(* IEC 61131-3 sources: std_i2980_v2.06_cp053/Source/IMM/ieccontrol/EjectorGeneral, 15 files *)

(* ---- FBConvertLintab.pu ---- *)
(*
@h    ! WARNING !
@h    The Kemro K2 system (including software) only meets category B according to EN 954-1,
@h    thus it is not intended for usage in safety-relevant control applications in the field
@h    of personal safety (e.g. emergency stop).
@h    To implement potentially necessary safety-relevant control tasks, always use additional
@h    external safety devices that are intended for the particular purpose, and meet the necessary
@h    functional safety.
@h    For further information see EN 954-1 (EN ISO 13849-1) and/or the K2-x00 user manual, chapter
@h    "CE conformity, directives and standards".

converts "relative" lintabs edited by the user into "absolute" linetabs used by the profile block.
difference between "absolute" and "relative" positions are limit offset and limit distance.

@FunctionID: S_KPIEC_PREJEC_EL_01
@FunctionID: A-ALLG-3

*)

IMPORT_OVER_LISTFILE
 TVisProfile
, FBChangeNoOfProfileSteps

END_IMPORT

FUNCTION_BLOCK FBConvertLintab #DUMMY_EDIT_BLOCK

VAR_INPUT
 bForward : BOOL (* forward or backward profile *);
END_VAR

VAR_IN_OUT
 LintabVis : TVisProfile (* "relative" lintab (displayed on hmi) *);
 LintabVisAbs : TVisProfile (* "absolute" lintab (for movement control) *);
END_VAR

VAR_INPUT
 rEjectorOfs : REAL (* offset between absolute and relative positions *);
 rEjectorDist : REAL (* max. ejector stroke *);
 bOpenEndProfile : BOOL := FALSE;
 bUseStartPosProfiles : BOOL;
 bDataStateIsReady : BOOL;
END_VAR

VAR_TEMP
 i : UDINT;
END_VAR

VAR
 rDif : REAL;
 fbChangeNoOfProfileSteps : FBChangeNoOfProfileSteps;
END_VAR
#BEGIN_EDIT_BLOCK
(**************************************** WARNING ********************************************
 *** The KEBA Kemro K2 System including software is not intended for safety control tasks! ***
 ***                       For further information see Comment tab!                        ***
 *********************************************************************************************)

// first element in fwd profile is 0
// first element in bwd profile is dist

fbChangeNoOfProfileSteps(ProfileVis := LintabVis,
                         bUseStartPosProfiles := bUseStartPosProfiles,
                         bOpenEndProfile := bOpenEndProfile,
                         bDataStateIsReady := bDataStateIsReady);

IF NOT bForward THEN
   LintabVis.Points[1].rStartPos:=rEjectorDist;
END_IF;

// first check vis lintab for plausibility and correct all points out of range
FOR i:=1 TO LintabVis.iNoOfPoints+1 DO
   // points must not be equal, so use a minimum difference of 0.1 between 2 points!
   IF bForward THEN
      rDif:=UDINT_TO_REAL((LintabVis.iNoOfPoints+1-i))*0.1;
   ELSE
      rDif:=UDINT_TO_REAL((i-1))*0.1;
   END_IF;
   LintabVis.Points[i].rStartPos:=MIN(LintabVis.Points[i].rStartPos, rEjectorDist - rDif);
END_FOR;

// copy lintab values
LintabVisAbs.iNoOfPoints:=LintabVis.iNoOfPoints;
LintabVisAbs.Points:=LintabVis.Points;

// calc absolute lintab, plausibility must be guaranteed by hmi
LintabVisAbs.iNoOfPoints:=LintabVis.iNoOfPoints;
FOR i:=1 TO LintabVis.iNoOfPoints+1 DO
  LintabVisAbs.Points[i].rStartPos:=LintabVis.Points[i].rStartPos+rEjectorOfs;
END_FOR;

;#END_EDIT_BLOCK END_FUNCTION_BLOCK

#END_OF_IEC_PART

@Puma @IecEditor 6 103 @Pou 25
@@@BEG_Comment@@@
@h    ! WARNING !
@h    The Kemro K2 system (including software) only meets category B according to EN 954-1,
@h    thus it is not intended for usage in safety-relevant control applications in the field
@h    of personal safety (e.g. emergency stop).
@h    To implement potentially necessary safety-relevant control tasks, always use additional
@h    external safety devices that are intended for the particular purpose, and meet the necessary
@h    functional safety.
@h    For further information see EN 954-1 (EN ISO 13849-1) and/or the K2-x00 user manual, chapter
@h    "CE conformity, directives and standards".

converts "relative" lintabs edited by the user into "absolute" linetabs used by the profile block.
difference between "absolute" and "relative" positions are limit offset and limit distance.

@FunctionID: S_KPIEC_PREJEC_EL_01
@FunctionID: A-ALLG-3

@@@END_Comment@@@

@BEG_Contents

@BEG_Func
@RT(17)FuncTreeContainer
0
@END_Func

@BEG_Const
@RT(18)ConstTreeContainer
0
@END_Const

@BEG_Export

@BEG_Kind
@FUNCTION_BLOCK @RT(15)FBConvertLintab @STRUCTURED_TEXT
@RT(0) @RT(0) @RT(0)
@END_Kind

@BEG_Dcl
@RT(16)DclTreeContainer
11
@Var @RT(8)bForward @RT(0) @T @F @DT @RT(4)BOOL @RT(0) @T @T @BASIC 0 @F
@F @F
@T
@BEG_Attrib
3 @RT(0) @RT(27)forward or backward profile @RT(0)
@END_Attrib
1 1 @F @F @F @F

@Var @RT(9)LintabVis @RT(0) @T @T @DERIVED 0 @T @T @DT @RT(11)TVisProfile @RT(0) @T @T @UNKNOWN 0 @F
@F @F
@T
@BEG_Attrib
3 @RT(0) @RT(36)"relative" lintab (displayed on hmi) @RT(0)
@END_Attrib
1 2 @F @F @F @F

@Var @RT(12)LintabVisAbs @RT(0) @T @T @DERIVED 0 @T @T @DT @RT(11)TVisProfile @RT(0) @T @T @UNKNOWN 0 @F
@F @F
@T
@BEG_Attrib
3 @RT(0) @RT(40)"absolute" lintab (for movement control) @RT(0)
@END_Attrib
1 2 @F @F @F @F

@Var @RT(11)rEjectorOfs @RT(0) @T @F @DT @RT(4)REAL @RT(0) @T @T @BASIC 0 @F
@F @F
@T
@BEG_Attrib
3 @RT(0) @RT(46)offset between absolute and relative positions @RT(0)
@END_Attrib
1 1 @F @F @F @F

@Var @RT(12)rEjectorDist @RT(0) @T @F @DT @RT(4)REAL @RT(0) @T @T @BASIC 0 @F
@F @F
@T
@BEG_Attrib
3 @RT(0) @RT(19)max. ejector stroke @RT(0)
@END_Attrib
1 1 @F @F @F @F

@Var @RT(15)bOpenEndProfile @RT(0) @T @F @DT @RT(4)BOOL @RT(0) @T @T @BASIC 0 @F
@F @F
@T
@BEG_Attrib
3 @RT(5)FALSE @RT(0) @RT(0)
@END_Attrib
1 1 @F @F @F @F

@Var @RT(20)bUseStartPosProfiles @RT(0) @T @F @DT @RT(4)BOOL @RT(0) @T @T @BASIC 0 @F
@F @F
@T
@BEG_Attrib
3 @RT(0) @RT(0) @RT(0)
@END_Attrib
1 1 @F @F @F @F

@Var @RT(17)bDataStateIsReady @RT(0) @T @F @DT @RT(4)BOOL @RT(0) @T @T @BASIC 0 @F
@F @F
@T
@BEG_Attrib
3 @RT(0) @RT(0) @RT(0)
@END_Attrib
1 1 @F @F @F @F

@Var @RT(1)i @RT(0) @T @F @DT @RT(5)UDINT @RT(0) @T @T @BASIC 0 @F
@F @F
@T
@BEG_Attrib
3 @RT(0) @RT(0) @RT(0)
@END_Attrib
1 4 @F @F @F @F

@Var @RT(4)rDif @RT(0) @T @F @DT @RT(4)REAL @RT(0) @T @T @BASIC 0 @F
@F @F
@T
@BEG_Attrib
3 @RT(0) @RT(0) @RT(0)
@END_Attrib
1 0 @F @F @F @F

@Var @RT(24)fbChangeNoOfProfileSteps @RT(0) @T @T @DERIVED 0 @T @T @DT @RT(24)FBChangeNoOfProfileSteps @RT(0) @T @T @UNKNOWN 0 @F
@F @F
@T
@BEG_Attrib
3 @RT(0) @RT(0) @RT(0)
@END_Attrib
1 0 @F @F @F @F

@END_Dcl

@END_Export

@BEG_Body
@TL(39)
(**************************************** WARNING ********************************************
 *** The KEBA Kemro K2 System including software is not intended for safety control tasks! ***
 ***                       For further information see Comment tab!                        ***
 *********************************************************************************************)

// first element in fwd profile is 0
// first element in bwd profile is dist

fbChangeNoOfProfileSteps(ProfileVis := LintabVis,
                         bUseStartPosProfiles := bUseStartPosProfiles,
                         bOpenEndProfile := bOpenEndProfile,
                         bDataStateIsReady := bDataStateIsReady);

IF NOT bForward THEN
   LintabVis.Points[1].rStartPos:=rEjectorDist;
END_IF;

// first check vis lintab for plausibility and correct all points out of range
FOR i:=1 TO LintabVis.iNoOfPoints+1 DO
   // points must not be equal, so use a minimum difference of 0.1 between 2 points!
   IF bForward THEN
      rDif:=UDINT_TO_REAL((LintabVis.iNoOfPoints+1-i))*0.1;
   ELSE
      rDif:=UDINT_TO_REAL((i-1))*0.1;
   END_IF;
   LintabVis.Points[i].rStartPos:=MIN(LintabVis.Points[i].rStartPos, rEjectorDist - rDif);
END_FOR;

// copy lintab values
LintabVisAbs.iNoOfPoints:=LintabVis.iNoOfPoints;
LintabVisAbs.Points:=LintabVis.Points;

// calc absolute lintab, plausibility must be guaranteed by hmi
LintabVisAbs.iNoOfPoints:=LintabVis.iNoOfPoints;
FOR i:=1 TO LintabVis.iNoOfPoints+1 DO
  LintabVisAbs.Points[i].rStartPos:=LintabVis.Points[i].rStartPos+rEjectorOfs;
END_FOR;

@END_Body

@END_Contents

(* ---- ABAdditionalEjectorSafety.pu ---- *)
(*
@h    ! WARNING !
@h    The Kemro K2 system (including software) only meets category B according to EN 954-1,
@h    thus it is not intended for usage in safety-relevant control applications in the field
@h    of personal safety (e.g. emergency stop).
@h    To implement potentially necessary safety-relevant control tasks, always use additional
@h    external safety devices that are intended for the particular purpose, and meet the necessary
@h    functional safety.
@h    For further information see EN 954-1 (EN ISO 13849-1) and/or the K2-x00 user manual, chapter
@h    "CE conformity, directives and standards".

AB for additional ejector safety.
- Lock mold close if monitor position is reached and ejector is not bwd
- resume mold close movement if ejector is bwd
- lock ejector fwd if mold position is lower or equal the ejector monitor position

- check ejector safety plate digin (mounted in the mold) if activated and
  lock all mold close movements if necessary.

@FunctionID: S_FU_02
*)

IMPORT_OVER_LISTFILE
 cCompMold
, IS_LINKED
, cMoveFwd
, tsDeviceId
, tnEjectorMode
, tevMovementState
, tnOperationMode
, tevMovementStateData
, FBLockUnlock
, FBLockUnlockGroup

END_IMPORT

ALGORITHM_BLOCK ABAdditionalEjectorSafety #DUMMY_EDIT_BLOCK

SYSTEM_VAR
 sv_bEjectorMonitorPos : BOOL (* ejector monitor position reached *);
 sv_rMoldPosition : REAL;
 sv_rEjectorMonitorPos : REAL (* ejector monitor position *);
 sv_bEjectorBwd : BOOL (* ejector is in bwd endposition *);
 sv_bEjectorFwd : BOOL (* ejector is in bwd endposition *);
 sv_DeviceId : tsDeviceId (* unique Device Identifier *);
 sv_bInitDone : BOOL;
 sv_EjectorMode : tnEjectorMode;
 sv_bOutputActive : BOOL (* Output is active *);
 sv_OperationMode : tnOperationMode;
 di_SafetyPlate : BOOL;
 sv_bCheckSafetyPlateDI : BOOL (* activates/deactivates the monitoring of di_SafetyPlate *);
 sv_bUseProgramSwitches : BOOL;
 sv_bOverrideEjectorSafety : BOOL;
END_VAR

SYSTEM_OBJECT
 TaskAnalog : TASK;
 EV_Task_3 : TASK;
 PU_Task_3 : TASK;
 evMovementState : tevMovementState;
 erEndPosChangedWithoutMove : ALARM;
 EV_Task_1 : TASK;
 erEjectorSafetyPlate : ALARM;
 erEjectorNotBackward : ALARM;
 erCompNotInCorrectPosition : ALARM;
END_OBJECT

VAR
 mevMovementState : tevMovementState;
END_VAR

PROCESS_ALGORITHM paCheckPosition ON TaskAnalog

#BEGIN_EDIT_BLOCK
(**************************************** WARNING ********************************************
 *** The KEBA Kemro K2 System including software is not intended for safety control tasks! ***
 ***                       For further information see Comment tab!                        ***
 *********************************************************************************************)

sv_bEjectorMonitorPos := (sv_rMoldPosition <= sv_rEjectorMonitorPos);

;#END_EDIT_BLOCK END_ALGORITHM

EVENT_ALGORITHM evaMovementState ON EV_Task_3 WITH mevMovementState

VAR_INPUT
 evMovementStateData : tevMovementStateData;
END_VAR
#BEGIN_EDIT_BLOCK
(**************************************** WARNING ********************************************
 *** The KEBA Kemro K2 System including software is not intended for safety control tasks! ***
 ***                       For further information see Comment tab!                        ***
 *********************************************************************************************)

//start/stop paCheckPosition
IF evMovementStateData.DeviceId.CompId <> cCompMold THEN
   RETURN;
END_IF;

IF evMovementStateData.State = nActive THEN
   IF sv_EjectorMode <> nNoUse AND sv_rEjectorMonitorPos <> 0.0 THEN
      //mold movement started and monitoring activated
      START_PROCESS_ALGORITHM(paCheckPosition);
   END_IF;
ELSE
   //mold movement stopped
   STOP_PROCESS_ALGORITHM(paCheckPosition);
END_IF;

;#END_EDIT_BLOCK END_ALGORITHM

POSTUPDATE_ALGORITHM pLockUnlockMoldAndEjector ON PU_Task_3 WITH sv_bEjectorMonitorPos,sv_bInitDone,sv_bEjectorBwd,sv_rEjectorMonitorPos,sv_EjectorMode,sv_bOverrideEjectorSafety,sv_bUseProgramSwitches

VAR
 fbLockUnlockMold : FBLockUnlock := (DeviceId:=(CompId:=cCompMold,IndexId:=1),MoveDir:=cMoveFwd,MoveId:=cMoveAll);
 fbLockUnlockEjector : FBLockUnlock := (DeviceId:=(CompId:=cCompEjector,IndexId:=1),MoveDir:=cMoveFwd,MoveId:=cMoveAll);
 fbLockUnlockGroup : FBLockUnlockGroup := (Group:=cLockGroupEjectorBwd);
 bInitDone : BOOL;
END_VAR
#BEGIN_EDIT_BLOCK
(**************************************** WARNING ********************************************
 *** The KEBA Kemro K2 System including software is not intended for safety control tasks! ***
 ***                       For further information see Comment tab!                        ***
 *********************************************************************************************)

IF sv_bUseProgramSwitches THEN
   mevMovementState := evMovementState;
ELSE
   mevMovementState := EMPTY;
END_IF;

IF NOT sv_bInitDone THEN
   //no lock/unlock events before init is done
   RETURN;
END_IF;

IF NOT bInitDone THEN
   fbLockUnlockMold.Alarm.AlarmId := erEjectorNotBackward;
   fbLockUnlockMold.Alarm.SubId[1] := 1; //only used to unify the alarm
   fbLockUnlockEjector.Alarm.AlarmId := erCompNotInCorrectPosition;
   fbLockUnlockEjector.Alarm.SubId[1] := cCompMold;
   fbLockUnlockEjector.Alarm.SubId[2] := 1;
   fbLockUnlockGroup.Alarm.AlarmId := erEjectorNotBackward;
   bInitDone := TRUE;
END_IF;

IF (sv_rEjectorMonitorPos = 0.0) OR NOT (sv_rMoldPosition <= sv_rEjectorMonitorPos) OR sv_bOverrideEjectorSafety OR NOT sv_bUseProgramSwitches THEN
   //unlock ejector fwd
   fbLockUnlockEjector.Mode := nUnlock;
ELSE
   //lock ejector fwd
   fbLockUnlockEjector.Mode := nLockResume;
END_IF;

IF (sv_EjectorMode = nNoUse) OR (sv_rEjectorMonitorPos = 0.0) OR NOT sv_bUseProgramSwitches THEN
   //ejector switched off or monitor position deactivated
   fbLockUnlockMold.Mode := nUnlock;
ELSIF (sv_rMoldPosition <= sv_rEjectorMonitorPos) AND NOT sv_bEjectorBwd THEN
   //monitor position reached and ejector not bwd -> lock mold fwd movement
   fbLockUnlockMold.Mode := nLockResume;
ELSIF sv_bEjectorBwd OR NOT (sv_rMoldPosition <= sv_rEjectorMonitorPos) THEN
   //ejector is bwd or monitor pos not reached -> unlock mold fwd movements
   fbLockUnlockMold.Mode := nUnlock;
END_IF;

//some movements are not allowed when ejector is not fully backward
IF sv_bEjectorBwd THEN
   fbLockUnlockGroup.Mode := nUnlock;
ELSE
   fbLockUnlockGroup.Mode := nLockAbort;
END_IF;

fbLockUnlockMold();
fbLockUnlockEjector();
fbLockUnlockGroup();

;#END_EDIT_BLOCK END_ALGORITHM

POSTUPDATE_ALGORITHM pEndPosChanged ON EV_Task_1 WITH sv_bEjectorBwd,sv_bEjectorFwd

#BEGIN_EDIT_BLOCK
(**************************************** WARNING ********************************************
 *** The KEBA Kemro K2 System including software is not intended for safety control tasks! ***
 ***                       For further information see Comment tab!                        ***
 *********************************************************************************************)

IF NOT sv_bInitDone OR (sv_OperationMode < nHalfAutomatic) THEN
   RETURN;
END_IF;

IF NOT sv_bOutputActive THEN
    SET_ALARM(Name := erEndPosChangedWithoutMove,
              SubID1 := sv_DeviceId.CompId,
              SubID2 := sv_DeviceId.IndexId);
END_IF;

;#END_EDIT_BLOCK END_ALGORITHM

POSTUPDATE_ALGORITHM pSafetyPlate ON PU_Task_3 WITH sv_bInitDone,sv_bCheckSafetyPlateDI,di_SafetyPlate

VAR
 bInitDone : BOOL;
 bSafetyPlateLinked : BOOL;
 fbLockUnlock : FBLockUnlock := (DeviceId:=(CompId:=cCompMold,IndexId:=1),MoveDir:=cMoveFwd,MoveId:=cMoveAll);
END_VAR
#BEGIN_EDIT_BLOCK
(**************************************** WARNING ********************************************
 *** The KEBA Kemro K2 System including software is not intended for safety control tasks! ***
 ***                       For further information see Comment tab!                        ***
 *********************************************************************************************)

IF NOT bInitDone THEN
   bSafetyPlateLinked := IS_LINKED(di_SafetyPlate);
   fbLockUnlock.DeviceId.CompId := cCompMold;
   fbLockUnlock.DeviceId.IndexId := 1;
   fbLockUnlock.MoveDir := cMoveFwd;
   fbLockUnlock.MoveId := cMoveAll;
   fbLockUnlock.Alarm.AlarmId := erEjectorSafetyPlate;
   fbLockUnlock.Alarm.SubId[1] := sv_DeviceId.IndexId;
   bInitDone := TRUE;
END_IF;

IF NOT sv_bInitDone OR NOT bSafetyPlateLinked THEN
   //init not done or no safety plate available
   RETURN;
END_IF;

IF sv_bCheckSafetyPlateDI THEN
   IF di_SafetyPlate THEN
      fbLockUnlock.Mode := nUnlock;
   ELSE
      fbLockUnlock.Mode := nLockAbort;
   END_IF;
ELSE
   //check deactivated -> unlock
   fbLockUnlock.Mode := nUnlock;
END_IF;

fbLockUnlock();

;#END_EDIT_BLOCK END_ALGORITHM

END_ALGORITHM_BLOCK

#END_OF_IEC_PART

@Puma @IecEditor 6 97 @Pou 25
@@@BEG_Comment@@@
@h    ! WARNING !
@h    The Kemro K2 system (including software) only meets category B according to EN 954-1,
@h    thus it is not intended for usage in safety-relevant control applications in the field
@h    of personal safety (e.g. emergency stop).
@h    To implement potentially necessary safety-relevant control tasks, always use additional
@h    external safety devices that are intended for the particular purpose, and meet the necessary
@h    functional safety.
@h    For further information see EN 954-1 (EN ISO 13849-1) and/or the K2-x00 user manual, chapter
@h    "CE conformity, directives and standards".

AB for additional ejector safety.
- Lock mold close if monitor position is reached and ejector is not bwd
- resume mold close movement if ejector is bwd
- lock ejector fwd if mold position is lower or equal the ejector monitor position

- check ejector safety plate digin (mounted in the mold) if activated and
  lock all mold close movements if necessary.

@FunctionID: S_FU_02
@@@END_Comment@@@

@BEG_Contents

@BEG_Func
@RT(17)FuncTreeContainer
2
@Var @RT(9)cCompMold @RT(0) @T @F @DT @RT(4)DINT @RT(0) @T @T @BASIC 0 @F
@F @F
@T
@BEG_Attrib
0 @RT(3)101 @RT(0)
@END_Attrib
1 1 @F @F @F @F

@Var @RT(9)IS_LINKED @RT(0) @T @T @DERIVED 0 @F @RT(22)KEBA_STANDARD_FUNCTION @F
@T
@BEG_Attrib
0 @RT(0) @RT(0)
@END_Attrib
1 1 @F @F @F @F

@END_Func

@BEG_Const
@RT(18)ConstTreeContainer
1
@Var @RT(8)cMoveFwd @RT(0) @T @F @DT @RT(4)DINT @RT(0) @T @T @BASIC 0 @F
@F @F
@T
@BEG_Attrib
0 @RT(2)12 @RT(16)movement forward
@END_Attrib
1 1 @F @F @F @F

@END_Const

@BEG_Export

@BEG_Kind
@ALGORITHM_BLOCK @RT(25)ABAdditionalEjectorSafety @STRUCTURED_TEXT
@RT(0) @RT(0) @RT(0)
@END_Kind

@BEG_Dcl
@RT(16)DclTreeContainer
24
@Var @RT(21)sv_bEjectorMonitorPos @RT(0) @T @F @DT @RT(4)BOOL @RT(0) @T @T @BASIC 0 @F
@F @F
@T
@BEG_Attrib
3 @RT(0) @RT(32)ejector monitor position reached @RT(0)
@END_Attrib
1 8 @F @F @F @F

@Var @RT(16)sv_rMoldPosition @RT(0) @T @F @DT @RT(4)REAL @RT(0) @T @T @BASIC 0 @F
@F @F
@T
@BEG_Attrib
3 @RT(0) @RT(0) @RT(0)
@END_Attrib
1 8 @F @F @F @F

@Var @RT(21)sv_rEjectorMonitorPos @RT(0) @T @F @DT @RT(4)REAL @RT(0) @T @T @BASIC 0 @F
@F @F
@T
@BEG_Attrib
3 @RT(0) @RT(24)ejector monitor position @RT(0)
@END_Attrib
1 8 @F @F @F @F

@Var @RT(14)sv_bEjectorBwd @RT(0) @T @F @DT @RT(4)BOOL @RT(0) @T @T @BASIC 0 @F
@F @F
@T
@BEG_Attrib
3 @RT(0) @RT(29)ejector is in bwd endposition @RT(0)
@END_Attrib
1 8 @F @F @F @F

@Var @RT(14)sv_bEjectorFwd @RT(0) @T @F @DT @RT(4)BOOL @RT(0) @T @T @BASIC 0 @F
@F @F
@T
@BEG_Attrib
3 @RT(0) @RT(29)ejector is in bwd endposition @RT(0)
@END_Attrib
1 8 @F @F @F @F

@Var @RT(11)sv_DeviceId @RT(0) @T @T @DERIVED 0 @T @T @DT @RT(10)tsDeviceId @RT(0) @T @T @UNKNOWN 0 @F
@F @F
@T
@BEG_Attrib
3 @RT(0) @RT(24)unique Device Identifier @RT(0)
@END_Attrib
1 8 @F @F @F @F

@Var @RT(12)sv_bInitDone @RT(0) @T @T @RENAMED 0 @T @T @DT @RT(4)BOOL @RT(0) @T @T @BASIC 0 @F
@F @F
@T
@BEG_Attrib
3 @RT(0) @RT(0) @RT(0)
@END_Attrib
1 8 @F @F @F @F

@Var @RT(14)sv_EjectorMode @RT(0) @T @T @DERIVED 0 @T @T @DT @RT(13)tnEjectorMode @RT(0) @T @T @UNKNOWN 0 @F
@F @F
@T
@BEG_Attrib
3 @RT(0) @RT(0) @RT(0)
@END_Attrib
1 8 @F @F @F @F

@Var @RT(16)sv_bOutputActive @RT(0) @T @F @DT @RT(4)BOOL @RT(0) @T @T @BASIC 0 @F
@F @F
@T
@BEG_Attrib
3 @RT(0) @RT(16)Output is active @RT(0)
@END_Attrib
1 8 @F @F @F @F

@Var @RT(10)TaskAnalog @RT(0) @T @F @DT @RT(4)TASK @RT(0) @T @T @BASIC 0 @F
@F @F
@T
@BEG_Attrib
3 @RT(0) @RT(0) @RT(0)
@END_Attrib
1 7 @F @F @F @F

@Var @RT(9)EV_Task_3 @RT(0) @T @F @DT @RT(4)TASK @RT(0) @T @T @BASIC 0 @F
@F @F
@T
@BEG_Attrib
3 @RT(0) @RT(0) @RT(0)
@END_Attrib
1 7 @F @F @F @F

@Var @RT(9)PU_Task_3 @RT(0) @T @F @DT @RT(4)TASK @RT(0) @T @T @BASIC 0 @F
@F @F
@T
@BEG_Attrib
3 @RT(0) @RT(0) @RT(0)
@END_Attrib
1 7 @F @F @F @F

@Var @RT(15)evMovementState @RT(0) @T @T @DERIVED 0 @T @T @DT @RT(16)tevMovementState @RT(0) @T @T @UNKNOWN 0 @F
@F @F
@T
@BEG_Attrib
3 @RT(0) @RT(0) @RT(0)
@END_Attrib
1 7 @F @F @F @F

@Var @RT(26)erEndPosChangedWithoutMove @RT(0) @T @F @DT @RT(5)ALARM @RT(0) @T @T @BASIC 0 @F
@F @F
@T
@BEG_Attrib
3 @RT(0) @RT(0) @RT(0)
@END_Attrib
1 7 @F @F @F @F

@Var @RT(9)EV_Task_1 @RT(0) @T @T @RENAMED 0 @T @T @DT @RT(4)TASK @RT(0) @T @T @BASIC 0 @F
@F @F
@T
@BEG_Attrib
3 @RT(0) @RT(0) @RT(0)
@END_Attrib
1 7 @F @F @F @F

@Var @RT(16)sv_OperationMode @RT(0) @T @T @DERIVED 0 @T @T @DT @RT(15)tnOperationMode @RT(0) @T @T @UNKNOWN 0 @F
@F @F
@T
@BEG_Attrib
3 @RT(0) @RT(0) @RT(0)
@END_Attrib
1 8 @F @F @F @F

@Var @RT(14)di_SafetyPlate @RT(0) @T @F @DT @RT(4)BOOL @RT(0) @T @T @BASIC 0 @F
@F @F
@T
@BEG_Attrib
3 @RT(0) @RT(0) @RT(0)
@END_Attrib
1 8 @F @F @F @F

@Var @RT(22)sv_bCheckSafetyPlateDI @RT(0) @T @F @DT @RT(4)BOOL @RT(0) @T @T @BASIC 0 @F
@F @F
@T
@BEG_Attrib
3 @RT(0) @RT(54)activates/deactivates the monitoring of di_SafetyPlate @RT(0)
@END_Attrib
1 8 @F @F @F @F

@Var @RT(20)erEjectorSafetyPlate @RT(0) @T @F @DT @RT(5)ALARM @RT(0) @T @T @BASIC 0 @F
@F @F
@T
@BEG_Attrib
3 @RT(0) @RT(0) @RT(0)
@END_Attrib
1 7 @F @F @F @F

@Var @RT(20)erEjectorNotBackward @RT(0) @T @T @RENAMED 0 @T @T @DT @RT(5)ALARM @RT(0) @T @T @BASIC 0 @F
@F @F
@T
@BEG_Attrib
3 @RT(0) @RT(0) @RT(0)
@END_Attrib
1 7 @F @F @F @F

@Var @RT(16)mevMovementState @RT(0) @T @T @RENAMED 0 @T @T @DT @RT(16)tevMovementState @RT(0) @T @T @UNKNOWN 0 @F
@F @F
@T
@BEG_Attrib
3 @RT(0) @RT(0) @RT(0)
@END_Attrib
1 0 @F @F @F @F

@Var @RT(22)sv_bUseProgramSwitches @RT(0) @T @F @DT @RT(4)BOOL @RT(0) @T @T @BASIC 0 @F
@F @F
@T
@BEG_Attrib
3 @RT(0) @RT(0) @RT(0)
@END_Attrib
1 8 @F @F @F @F

@Var @RT(25)sv_bOverrideEjectorSafety @RT(0) @T @F @DT @RT(4)BOOL @RT(0) @T @T @BASIC 0 @F
@F @F
@T
@BEG_Attrib
3 @RT(0) @RT(0) @RT(0)
@END_Attrib
1 8 @F @F @F @F

@Var @RT(26)erCompNotInCorrectPosition @RT(0) @T @F @DT @RT(5)ALARM @RT(0) @T @T @BASIC 0 @F
@F @F
@T
@BEG_Attrib
3 @RT(0) @RT(0) @RT(0)
@END_Attrib
1 7 @F @F @F @F

@END_Dcl

@END_Export

@BEG_Body

5

@BEG_Export

@BEG_Algo
@PROCESS_ALGORITHM @RT(15)paCheckPosition @STRUCTURED_TEXT
@RT(0) @RT(0) @RT(10)TaskAnalog @F @F
@END_Algo

@BEG_Dcl
@RT(16)DclTreeContainer
0
@END_Dcl

@END_Export

@BEG_Export

@BEG_Algo
@EVENT_ALGORITHM @RT(16)evaMovementState @STRUCTURED_TEXT
@RT(0) @RT(16)mevMovementState @RT(9)EV_Task_3 @F @F
@END_Algo

@BEG_Dcl
@RT(16)DclTreeContainer
1
@Var @RT(19)evMovementStateData @RT(0) @T @T @DERIVED 0 @T @T @DT @RT(20)tevMovementStateData @RT(0) @T @T @UNKNOWN 0 @F
@F @F
@T
@BEG_Attrib
3 @RT(0) @RT(0) @RT(0)
@END_Attrib
1 1 @F @F @F @F

@END_Dcl

@END_Export

@BEG_Export

@BEG_Algo
@POSTUPDATE_ALGORITHM @RT(25)pLockUnlockMoldAndEjector @STRUCTURED_TEXT
@RT(0) @RT(135)sv_bEjectorMonitorPos,sv_bInitDone,sv_bEjectorBwd,sv_rEjectorMonitorPos,sv_EjectorMode,sv_bOverrideEjectorSafety,sv_bUseProgramSwitches @RT(9)PU_Task_3 @F @F
@END_Algo

@BEG_Dcl
@RT(16)DclTreeContainer
4
@Var @RT(16)fbLockUnlockMold @RT(0) @T @T @DERIVED 0 @T @T @DT @RT(12)FBLockUnlock @RT(0) @T @T @UNKNOWN 0 @F
@F @F
@T
@BEG_Attrib
3 @RT(77)(DeviceId:=(CompId:=cCompMold,IndexId:=1),MoveDir:=cMoveFwd,MoveId:=cMoveAll) @RT(0) @RT(0)
@END_Attrib
1 0 @F @F @F @F

@Var @RT(19)fbLockUnlockEjector @RT(0) @T @T @DERIVED 0 @T @T @DT @RT(12)FBLockUnlock @RT(0) @T @T @UNKNOWN 0 @F
@F @F
@T
@BEG_Attrib
3 @RT(80)(DeviceId:=(CompId:=cCompEjector,IndexId:=1),MoveDir:=cMoveFwd,MoveId:=cMoveAll) @RT(0) @RT(0)
@END_Attrib
1 0 @F @F @F @F

@Var @RT(17)fbLockUnlockGroup @RT(0) @T @T @DERIVED 0 @T @T @DT @RT(17)FBLockUnlockGroup @RT(0) @T @T @UNKNOWN 0 @F
@F @F
@T
@BEG_Attrib
3 @RT(29)(Group:=cLockGroupEjectorBwd) @RT(0) @RT(0)
@END_Attrib
1 0 @F @F @F @F

@Var @RT(9)bInitDone @RT(0) @T @F @DT @RT(4)BOOL @RT(0) @T @T @BASIC 0 @F
@F @F
@T
@BEG_Attrib
3 @RT(0) @RT(0) @RT(0)
@END_Attrib
1 0 @F @F @F @F

@END_Dcl

@END_Export

@BEG_Export

@BEG_Algo
@POSTUPDATE_ALGORITHM @RT(14)pEndPosChanged @STRUCTURED_TEXT
@RT(0) @RT(29)sv_bEjectorBwd,sv_bEjectorFwd @RT(9)EV_Task_1 @F @F
@END_Algo

@BEG_Dcl
@RT(16)DclTreeContainer
0
@END_Dcl

@END_Export

@BEG_Export

@BEG_Algo
@POSTUPDATE_ALGORITHM @RT(12)pSafetyPlate @STRUCTURED_TEXT
@RT(0) @RT(50)sv_bInitDone,sv_bCheckSafetyPlateDI,di_SafetyPlate @RT(9)PU_Task_3 @F @F
@END_Algo

@BEG_Dcl
@RT(16)DclTreeContainer
3
@Var @RT(9)bInitDone @RT(0) @T @F @DT @RT(4)BOOL @RT(0) @T @T @BASIC 0 @F
@F @F
@T
@BEG_Attrib
3 @RT(0) @RT(0) @RT(0)
@END_Attrib
1 0 @F @F @F @F

@Var @RT(18)bSafetyPlateLinked @RT(0) @T @F @DT @RT(4)BOOL @RT(0) @T @T @BASIC 0 @F
@F @F
@T
@BEG_Attrib
3 @RT(0) @RT(0) @RT(0)
@END_Attrib
1 0 @F @F @F @F

@Var @RT(12)fbLockUnlock @RT(0) @T @T @DERIVED 0 @T @T @DT @RT(12)FBLockUnlock @RT(0) @T @T @UNKNOWN 0 @F
@F @F
@T
@BEG_Attrib
3 @RT(77)(DeviceId:=(CompId:=cCompMold,IndexId:=1),MoveDir:=cMoveFwd,MoveId:=cMoveAll) @RT(0) @RT(0)
@END_Attrib
1 0 @F @F @F @F

@END_Dcl

@END_Export

@BEG_Body
@TL(7)
(**************************************** WARNING ********************************************
 *** The KEBA Kemro K2 System including software is not intended for safety control tasks! ***
 ***                       For further information see Comment tab!                        ***
 *********************************************************************************************)

sv_bEjectorMonitorPos := (sv_rMoldPosition <= sv_rEjectorMonitorPos);

@END_Body

@@@BEG_Comment@@@
@TL(0)

@@@END_Comment@@@

@BEG_Body
@TL(20)
(**************************************** WARNING ********************************************
 *** The KEBA Kemro K2 System including software is not intended for safety control tasks! ***
 ***                       For further information see Comment tab!                        ***
 *********************************************************************************************)

//start/stop paCheckPosition
IF evMovementStateData.DeviceId.CompId <> cCompMold THEN
   RETURN;
END_IF;

IF evMovementStateData.State = nActive THEN
   IF sv_EjectorMode <> nNoUse AND sv_rEjectorMonitorPos <> 0.0 THEN
      //mold movement started and monitoring activated
      START_PROCESS_ALGORITHM(paCheckPosition);
   END_IF;
ELSE
   //mold movement stopped
   STOP_PROCESS_ALGORITHM(paCheckPosition);
END_IF;

@END_Body

@@@BEG_Comment@@@
@TL(0)

@@@END_Comment@@@

@BEG_Body
@TL(57)
(**************************************** WARNING ********************************************
 *** The KEBA Kemro K2 System including software is not intended for safety control tasks! ***
 ***                       For further information see Comment tab!                        ***
 *********************************************************************************************)

IF sv_bUseProgramSwitches THEN
   mevMovementState := evMovementState;
ELSE
   mevMovementState := EMPTY;
END_IF;

IF NOT sv_bInitDone THEN
   //no lock/unlock events before init is done
   RETURN;
END_IF;

IF NOT bInitDone THEN
   fbLockUnlockMold.Alarm.AlarmId := erEjectorNotBackward;
   fbLockUnlockMold.Alarm.SubId[1] := 1; //only used to unify the alarm
   fbLockUnlockEjector.Alarm.AlarmId := erCompNotInCorrectPosition;
   fbLockUnlockEjector.Alarm.SubId[1] := cCompMold;
   fbLockUnlockEjector.Alarm.SubId[2] := 1;
   fbLockUnlockGroup.Alarm.AlarmId := erEjectorNotBackward;
   bInitDone := TRUE;
END_IF;

IF (sv_rEjectorMonitorPos = 0.0) OR NOT (sv_rMoldPosition <= sv_rEjectorMonitorPos) OR sv_bOverrideEjectorSafety OR NOT sv_bUseProgramSwitches THEN
   //unlock ejector fwd
   fbLockUnlockEjector.Mode := nUnlock;
ELSE
   //lock ejector fwd
   fbLockUnlockEjector.Mode := nLockResume;
END_IF;

IF (sv_EjectorMode = nNoUse) OR (sv_rEjectorMonitorPos = 0.0) OR NOT sv_bUseProgramSwitches THEN
   //ejector switched off or monitor position deactivated
   fbLockUnlockMold.Mode := nUnlock;
ELSIF (sv_rMoldPosition <= sv_rEjectorMonitorPos) AND NOT sv_bEjectorBwd THEN
   //monitor position reached and ejector not bwd -> lock mold fwd movement
   fbLockUnlockMold.Mode := nLockResume;
ELSIF sv_bEjectorBwd OR NOT (sv_rMoldPosition <= sv_rEjectorMonitorPos) THEN
   //ejector is bwd or monitor pos not reached -> unlock mold fwd movements
   fbLockUnlockMold.Mode := nUnlock;
END_IF;

//some movements are not allowed when ejector is not fully backward
IF sv_bEjectorBwd THEN
   fbLockUnlockGroup.Mode := nUnlock;
ELSE
   fbLockUnlockGroup.Mode := nLockAbort;
END_IF;

fbLockUnlockMold();
fbLockUnlockEjector();
fbLockUnlockGroup();

@END_Body

@@@BEG_Comment@@@
@TL(0)

@@@END_Comment@@@

@BEG_Body
@TL(15)
(**************************************** WARNING ********************************************
 *** The KEBA Kemro K2 System including software is not intended for safety control tasks! ***
 ***                       For further information see Comment tab!                        ***
 *********************************************************************************************)

IF NOT sv_bInitDone OR (sv_OperationMode < nHalfAutomatic) THEN
   RETURN;
END_IF;

IF NOT sv_bOutputActive THEN
    SET_ALARM(Name := erEndPosChangedWithoutMove,
              SubID1 := sv_DeviceId.CompId,
              SubID2 := sv_DeviceId.IndexId);
END_IF;

@END_Body

@@@BEG_Comment@@@
@TL(0)

@@@END_Comment@@@

@BEG_Body
@TL(36)
(**************************************** WARNING ********************************************
 *** The KEBA Kemro K2 System including software is not intended for safety control tasks! ***
 ***                       For further information see Comment tab!                        ***
 *********************************************************************************************)

IF NOT bInitDone THEN
   bSafetyPlateLinked := IS_LINKED(di_SafetyPlate);
   fbLockUnlock.DeviceId.CompId := cCompMold;
   fbLockUnlock.DeviceId.IndexId := 1;
   fbLockUnlock.MoveDir := cMoveFwd;
   fbLockUnlock.MoveId := cMoveAll;
   fbLockUnlock.Alarm.AlarmId := erEjectorSafetyPlate;
   fbLockUnlock.Alarm.SubId[1] := sv_DeviceId.IndexId;
   bInitDone := TRUE;
END_IF;

IF NOT sv_bInitDone OR NOT bSafetyPlateLinked THEN
   //init not done or no safety plate available
   RETURN;
END_IF;

IF sv_bCheckSafetyPlateDI THEN
   IF di_SafetyPlate THEN
      fbLockUnlock.Mode := nUnlock;
   ELSE
      fbLockUnlock.Mode := nLockAbort;
   END_IF;
ELSE
   //check deactivated -> unlock
   fbLockUnlock.Mode := nUnlock;
END_IF;

fbLockUnlock();

@END_Body

@@@BEG_Comment@@@
@TL(0)

@@@END_Comment@@@
@END_Body

@END_Contents

(* ---- ABButtonControl.pu ---- *)
IMPORT_OVER_LISTFILE
 IS_LINKED
, ABManualButton
, tevPanelButtonRegister
, tsDeviceId
, tyPanelButton
, tevPanelButtonRegisterData
, tsPanelButton

END_IMPORT

ALGORITHM_BLOCK ABButtonControl #DUMMY_EDIT_BLOCK

SYSTEM_VAR
 sv_bTransducerAvailable : BOOL;
 sv_DeviceId : tsDeviceId;
 sv_bDeviceReady : BOOL;
 sv_bEjectorBwd : BOOL;
 sv_bEjectorFwd : BOOL;
 sv_bInitStart : BOOL;
 sv_rEjectorStroke : REAL;
 sv_rEjectorPositionRel : REAL;
 sv_iPanelMovementSelector : DINT;
 sv_PanelButtons : tyPanelButton;
 di_ButtonFwd : BOOL;
 di_ButtonBwd : BOOL;
 di_ButtonGeneral1 : BOOL;
 di_ButtonGeneral2 : BOOL;
 sv_bButtonFwd : BOOL;
 sv_bButtonBwd : BOOL;
END_VAR

SYSTEM_OBJECT
 PU_Task_13 : TASK;
 PU_Task_7 : TASK;
 evPanelButtonRegister : tevPanelButtonRegister;
END_OBJECT

VAR
 abManualButton : ABManualButton;
 evPanelButtonRegisterData : tevPanelButtonRegisterData;
 mbDIButtonFwdLinked : BOOL;
 mbDIButtonBwdLinked : BOOL;
 mbDIButtonGeneralFwdLinked : BOOL;
 mbDIButtonGeneralBwdLinked : BOOL;
 mpbButtonGeneralFwd : REFTO BOOL;
 mpbButtonGeneralBwd : REFTO BOOL;
 mpiPanelMovementSelector : REFTO DINT;
END_VAR

VAR CONSTANT
 cButtonMoveFwdBwd : DINT := 1;
END_VAR

POSTUPDATE_ALGORITHM pRegisterButtons ON PU_Task_13 WITH sv_bInitStart

#BEGIN_EDIT_BLOCK
(**************************************** WARNING ********************************************
 *** The KEBA Kemro K2 System including software is not intended for safety control tasks! ***
 ***                       For further information see Comment tab!                        ***
 *********************************************************************************************)

mpbButtonGeneralFwd := EMPTY;
mpbButtonGeneralBwd := EMPTY;

mbDIButtonFwdLinked := IS_LINKED(di_ButtonFwd);
mbDIButtonBwdLinked := IS_LINKED(di_ButtonBwd);

mbDIButtonGeneralFwdLinked := IS_LINKED(di_ButtonGeneral2);
mbDIButtonGeneralBwdLinked := IS_LINKED(di_ButtonGeneral1);

IF (mbDIButtonGeneralFwdLinked AND mbDIButtonGeneralBwdLinked) THEN
    mpiPanelMovementSelector := @sv_iPanelMovementSelector;
END_IF;

// register combinded fwd/bwd button
evPanelButtonRegisterData.Button.nPanelButtonType := nPanelButtonMovement;
evPanelButtonRegisterData.Button.iCompId := sv_DeviceId.CompId;
evPanelButtonRegisterData.Button.iIndexId := sv_DeviceId.IndexId;
evPanelButtonRegisterData.Button.iButtonId := cButtonMoveFwdBwd;
evPanelButtonRegisterData.Button.pbActionVar1 := @sv_bButtonBwd;
evPanelButtonRegisterData.Button.pbActionVar2 := @sv_bButtonFwd;
evPanelButtonRegisterData.Button.Optional.pbLimitSwitch1:= @sv_bEjectorBwd;
evPanelButtonRegisterData.Button.Optional.pbLimitSwitch2:= @sv_bEjectorFwd;
IF sv_bTransducerAvailable THEN
   evPanelButtonRegisterData.Button.Optional.prActVar := @sv_rEjectorPositionRel;
END_IF;
evPanelButtonRegisterData.Button.Optional.prMaxVar := @sv_rEjectorStroke;
evPanelButtonRegisterData.Button.Optional.prMinVar := EMPTY;
evPanelButtonRegisterData.Button.Optional.iBarAttr := 0;

SET_EVENT(evPanelButtonRegister, evPanelButtonRegisterData);

;#END_EDIT_BLOCK END_ALGORITHM

POSTUPDATE_ALGORITHM pButtonFwd ON PU_Task_7 WITH di_ButtonFwd,sv_bButtonFwd,mpbButtonGeneralFwd^

VAR
 bButton : BOOL;
END_VAR
#BEGIN_EDIT_BLOCK
(**************************************** WARNING ********************************************
 *** The KEBA Kemro K2 System including software is not intended for safety control tasks! ***
 ***                       For further information see Comment tab!                        ***
 *********************************************************************************************)

// soft panel button
bButton := sv_bButtonFwd;

// hw panel button
IF mbDIButtonFwdLinked THEN
    bButton := bButton OR di_ButtonFwd;
END_IF;

// external panel button
IF CHECK_REF(mpbButtonGeneralFwd^) THEN
    bButton := bButton OR mpbButtonGeneralFwd^;
END_IF;

abManualButton.aButtonFwd(bButtonFwd := bButton);

;#END_EDIT_BLOCK END_ALGORITHM

POSTUPDATE_ALGORITHM pButtonBwd ON PU_Task_7 WITH di_ButtonBwd,sv_bButtonBwd,mpbButtonGeneralBwd^

VAR
 bButton : BOOL;
END_VAR
#BEGIN_EDIT_BLOCK
(**************************************** WARNING ********************************************
 *** The KEBA Kemro K2 System including software is not intended for safety control tasks! ***
 ***                       For further information see Comment tab!                        ***
 *********************************************************************************************)

// soft panel button
bButton := sv_bButtonBwd;

// hw panel button
IF mbDIButtonBwdLinked THEN
    bButton := bButton OR di_ButtonBwd;
END_IF;

// external panel button
IF CHECK_REF(mpbButtonGeneralBwd^) THEN
    bButton := bButton OR mpbButtonGeneralBwd^;
END_IF;

abManualButton.aButtonBwd(bButtonBwd := bButton);

;#END_EDIT_BLOCK END_ALGORITHM

POSTUPDATE_ALGORITHM pMoveSelectorChanged ON PU_Task_7 WITH mpiPanelMovementSelector^

VAR
 Button : tsPanelButton;
END_VAR
#BEGIN_EDIT_BLOCK
(**************************************** WARNING ********************************************
 *** The KEBA Kemro K2 System including software is not intended for safety control tasks! ***
 ***                       For further information see Comment tab!                        ***
 *********************************************************************************************)
mpbButtonGeneralFwd := EMPTY;
mpbButtonGeneralBwd := EMPTY;

IF (NOT sv_bDeviceReady) THEN
    // stop active movements
    abManualButton.aButtonFwd(bButtonFwd := FALSE);
    abManualButton.aButtonBwd(bButtonBwd := FALSE);
END_IF;

IF (sv_iPanelMovementSelector > 0) THEN
    Button := sv_PanelButtons[sv_iPanelMovementSelector];
    IF (Button.iCompId = sv_DeviceId.CompId AND
        Button.iIndexId = sv_DeviceId.IndexId) THEN
        IF (Button.iButtonId = cButtonMoveFwdBwd) THEN
            mpbButtonGeneralFwd := @di_ButtonGeneral2;
            mpbButtonGeneralBwd := @di_ButtonGeneral1;
        END_IF;
    END_IF;
END_IF;

;#END_EDIT_BLOCK END_ALGORITHM

END_ALGORITHM_BLOCK

#END_OF_IEC_PART

@Puma @IecEditor 6 150 @Pou 25
@@@BEG_Comment@@@

@@@END_Comment@@@

@BEG_Contents

@BEG_Func
@RT(17)FuncTreeContainer
1
@Var @RT(9)IS_LINKED @RT(0) @T @T @DERIVED 0 @F @RT(22)KEBA_STANDARD_FUNCTION @F
@T
@BEG_Attrib
0 @RT(0) @RT(0)
@END_Attrib
1 1 @F @F @F @F

@END_Func

@BEG_Const
@RT(18)ConstTreeContainer
0
@END_Const

@BEG_Export

@BEG_Kind
@ALGORITHM_BLOCK @RT(15)ABButtonControl @STRUCTURED_TEXT
@RT(0) @RT(0) @RT(0)
@END_Kind

@BEG_Dcl
@RT(16)DclTreeContainer
29
@Var @RT(14)abManualButton @RT(0) @T @T @DERIVED 0 @T @T @DT @RT(14)ABManualButton @RT(0) @T @T @UNKNOWN 0 @F
@F @F
@T
@BEG_Attrib
3 @RT(0) @RT(0) @RT(0)
@END_Attrib
1 0 @F @F @F @F

@Var @RT(10)PU_Task_13 @RT(0) @T @T @RENAMED 0 @T @T @DT @RT(4)TASK @RT(0) @T @T @BASIC 0 @F
@F @F
@T
@BEG_Attrib
3 @RT(0) @RT(0) @RT(0)
@END_Attrib
1 7 @F @F @F @F

@Var @RT(9)PU_Task_7 @RT(0) @T @T @RENAMED 0 @T @T @DT @RT(4)TASK @RT(0) @T @T @BASIC 0 @F
@F @F
@T
@BEG_Attrib
3 @RT(0) @RT(0) @RT(0)
@END_Attrib
1 7 @F @F @F @F

@Var @RT(23)sv_bTransducerAvailable @RT(0) @T @F @DT @RT(4)BOOL @RT(0) @T @T @BASIC 0 @F
@F @F
@T
@BEG_Attrib
3 @RT(0) @RT(0) @RT(0)
@END_Attrib
1 8 @F @F @F @F

@Var @RT(21)evPanelButtonRegister @RT(0) @T @T @DERIVED 0 @T @T @DT @RT(22)tevPanelButtonRegister @RT(0) @T @T @UNKNOWN 0 @F
@F @F
@T
@BEG_Attrib
3 @RT(0) @RT(0) @RT(0)
@END_Attrib
1 7 @F @F @F @F

@Var @RT(11)sv_DeviceId @RT(0) @T @T @DERIVED 0 @T @T @DT @RT(10)tsDeviceId @RT(0) @T @T @UNKNOWN 0 @F
@F @F
@T
@BEG_Attrib
3 @RT(0) @RT(0) @RT(0)
@END_Attrib
1 8 @F @F @F @F

@Var @RT(15)sv_bDeviceReady @RT(0) @T @T @RENAMED 0 @T @T @DT @RT(4)BOOL @RT(0) @T @T @BASIC 0 @F
@F @F
@T
@BEG_Attrib
3 @RT(0) @RT(0) @RT(0)
@END_Attrib
1 8 @F @F @F @F

@Var @RT(14)sv_bEjectorBwd @RT(0) @T @T @RENAMED 0 @T @T @DT @RT(4)BOOL @RT(0) @T @T @BASIC 0 @F
@F @F
@T
@BEG_Attrib
3 @RT(0) @RT(0) @RT(0)
@END_Attrib
1 8 @F @F @F @F

@Var @RT(14)sv_bEjectorFwd @RT(0) @T @T @RENAMED 0 @T @T @DT @RT(4)BOOL @RT(0) @T @T @BASIC 0 @F
@F @F
@T
@BEG_Attrib
3 @RT(0) @RT(0) @RT(0)
@END_Attrib
1 8 @F @F @F @F

@Var @RT(13)sv_bInitStart @RT(0) @T @T @RENAMED 0 @T @T @DT @RT(4)BOOL @RT(0) @T @T @BASIC 0 @F
@F @F
@T
@BEG_Attrib
3 @RT(0) @RT(0) @RT(0)
@END_Attrib
1 8 @F @F @F @F

@Var @RT(17)sv_rEjectorStroke @RT(0) @T @F @DT @RT(4)REAL @RT(0) @T @T @BASIC 0 @F
@F @F
@T
@BEG_Attrib
3 @RT(0) @RT(0) @RT(0)
@END_Attrib
1 8 @F @F @F @F

@Var @RT(22)sv_rEjectorPositionRel @RT(0) @T @F @DT @RT(4)REAL @RT(0) @T @T @BASIC 0 @F
@F @F
@T
@BEG_Attrib
3 @RT(0) @RT(0) @RT(0)
@END_Attrib
1 8 @F @F @F @F

@Var @RT(25)sv_iPanelMovementSelector @RT(0) @T @F @DT @RT(4)DINT @RT(0) @T @T @BASIC 0 @F
@F @F
@T
@BEG_Attrib
3 @RT(0) @RT(0) @RT(0)
@END_Attrib
1 8 @F @F @F @F

@Var @RT(15)sv_PanelButtons @RT(0) @T @T @DERIVED 0 @T @T @DT @RT(13)tyPanelButton @RT(0) @T @T @UNKNOWN 0 @F
@F @F
@T
@BEG_Attrib
3 @RT(0) @RT(0) @RT(0)
@END_Attrib
1 8 @F @F @F @F

@Var @RT(12)di_ButtonFwd @RT(0) @T @T @RENAMED 0 @T @T @DT @RT(4)BOOL @RT(0) @T @T @BASIC 0 @F
@F @F
@T
@BEG_Attrib
3 @RT(0) @RT(0) @RT(0)
@END_Attrib
1 8 @F @F @F @F

@Var @RT(12)di_ButtonBwd @RT(0) @T @T @RENAMED 0 @T @T @DT @RT(4)BOOL @RT(0) @T @T @BASIC 0 @F
@F @F
@T
@BEG_Attrib
3 @RT(0) @RT(0) @RT(0)
@END_Attrib
1 8 @F @F @F @F

@Var @RT(17)di_ButtonGeneral1 @RT(0) @T @F @DT @RT(4)BOOL @RT(0) @T @T @BASIC 0 @F
@F @F
@T
@BEG_Attrib
3 @RT(0) @RT(0) @RT(0)
@END_Attrib
1 8 @F @F @F @F

@Var @RT(17)di_ButtonGeneral2 @RT(0) @T @F @DT @RT(4)BOOL @RT(0) @T @T @BASIC 0 @F
@F @F
@T
@BEG_Attrib
3 @RT(0) @RT(0) @RT(0)
@END_Attrib
1 8 @F @F @F @F

@Var @RT(13)sv_bButtonFwd @RT(0) @T @F @DT @RT(4)BOOL @RT(0) @T @T @BASIC 0 @F
@F @F
@T
@BEG_Attrib
3 @RT(0) @RT(0) @RT(0)
@END_Attrib
1 8 @F @F @F @F

@Var @RT(13)sv_bButtonBwd @RT(0) @T @F @DT @RT(4)BOOL @RT(0) @T @T @BASIC 0 @F
@F @F
@T
@BEG_Attrib
3 @RT(0) @RT(0) @RT(0)
@END_Attrib
1 8 @F @F @F @F

@Var @RT(17)cButtonMoveFwdBwd @RT(0) @T @F @DT @RT(4)DINT @RT(0) @T @T @BASIC 0 @F
@F @F
@T
@BEG_Attrib
3 @RT(1)1 @RT(0) @RT(0)
@END_Attrib
1 15 @F @F @F @F

@Var @RT(25)evPanelButtonRegisterData @RT(0) @T @T @DERIVED 0 @T @T @DT @RT(26)tevPanelButtonRegisterData @RT(0) @T @T @UNKNOWN 0 @F
@F @F
@T
@BEG_Attrib
3 @RT(0) @RT(0) @RT(0)
@END_Attrib
1 0 @F @F @F @F

@Var @RT(19)mbDIButtonFwdLinked @RT(0) @T @T @RENAMED 0 @T @T @DT @RT(4)BOOL @RT(0) @T @T @BASIC 0 @F
@F @F
@T
@BEG_Attrib
3 @RT(0) @RT(0) @RT(0)
@END_Attrib
1 0 @F @F @F @F

@Var @RT(19)mbDIButtonBwdLinked @RT(0) @T @T @RENAMED 0 @T @T @DT @RT(4)BOOL @RT(0) @T @T @BASIC 0 @F
@F @F
@T
@BEG_Attrib
3 @RT(0) @RT(0) @RT(0)
@END_Attrib
1 0 @F @F @F @F

@Var @RT(26)mbDIButtonGeneralFwdLinked @RT(0) @T @T @RENAMED 0 @T @T @DT @RT(4)BOOL @RT(0) @T @T @BASIC 0 @F
@F @F
@T
@BEG_Attrib
3 @RT(0) @RT(0) @RT(0)
@END_Attrib
1 0 @F @F @F @F

@Var @RT(26)mbDIButtonGeneralBwdLinked @RT(0) @T @T @RENAMED 0 @T @T @DT @RT(4)BOOL @RT(0) @T @T @BASIC 0 @F
@F @F
@T
@BEG_Attrib
3 @RT(0) @RT(0) @RT(0)
@END_Attrib
1 0 @F @F @F @F

@Var @RT(19)mpbButtonGeneralFwd @RT(0) @T @T @REFTO 0 @T @DT @RT(4)BOOL @RT(0) @T @T @BASIC 0 @F
@F @F
@T
@BEG_Attrib
3 @RT(0) @RT(0) @RT(0)
@END_Attrib
1 0 @F @F @F @F

@Var @RT(19)mpbButtonGeneralBwd @RT(0) @T @T @REFTO 0 @T @DT @RT(4)BOOL @RT(0) @T @T @BASIC 0 @F
@F @F
@T
@BEG_Attrib
3 @RT(0) @RT(0) @RT(0)
@END_Attrib
1 0 @F @F @F @F

@Var @RT(24)mpiPanelMovementSelector @RT(0) @T @T @REFTO 0 @T @DT @RT(4)DINT @RT(0) @T @T @BASIC 0 @F
@F @F
@T
@BEG_Attrib
3 @RT(0) @RT(0) @RT(0)
@END_Attrib
1 0 @F @F @F @F

@END_Dcl

@END_Export

@BEG_Body

4

@BEG_Export

@BEG_Algo
@POSTUPDATE_ALGORITHM @RT(16)pRegisterButtons @STRUCTURED_TEXT
@RT(0) @RT(13)sv_bInitStart @RT(10)PU_Task_13 @F @F
@END_Algo

@BEG_Dcl
@RT(16)DclTreeContainer
0
@END_Dcl

@END_Export

@BEG_Export

@BEG_Algo
@POSTUPDATE_ALGORITHM @RT(10)pButtonFwd @STRUCTURED_TEXT
@RT(0) @RT(47)di_ButtonFwd,sv_bButtonFwd,mpbButtonGeneralFwd^ @RT(9)PU_Task_7 @F @F
@END_Algo

@BEG_Dcl
@RT(16)DclTreeContainer
1
@Var @RT(7)bButton @RT(0) @T @F @DT @RT(4)BOOL @RT(0) @T @T @BASIC 0 @F
@F @F
@T
@BEG_Attrib
3 @RT(0) @RT(0) @RT(0)
@END_Attrib
1 0 @F @F @F @F

@END_Dcl

@END_Export

@BEG_Export

@BEG_Algo
@POSTUPDATE_ALGORITHM @RT(10)pButtonBwd @STRUCTURED_TEXT
@RT(0) @RT(47)di_ButtonBwd,sv_bButtonBwd,mpbButtonGeneralBwd^ @RT(9)PU_Task_7 @F @F
@END_Algo

@BEG_Dcl
@RT(16)DclTreeContainer
1
@Var @RT(7)bButton @RT(0) @T @F @DT @RT(4)BOOL @RT(0) @T @T @BASIC 0 @F
@F @F
@T
@BEG_Attrib
3 @RT(0) @RT(0) @RT(0)
@END_Attrib
1 0 @F @F @F @F

@END_Dcl

@END_Export

@BEG_Export

@BEG_Algo
@POSTUPDATE_ALGORITHM @RT(20)pMoveSelectorChanged @STRUCTURED_TEXT
@RT(0) @RT(25)mpiPanelMovementSelector^ @RT(9)PU_Task_7 @F @F
@END_Algo

@BEG_Dcl
@RT(16)DclTreeContainer
1
@Var @RT(6)Button @RT(0) @T @T @DERIVED 0 @T @T @DT @RT(13)tsPanelButton @RT(0) @T @T @UNKNOWN 0 @F
@F @F
@T
@BEG_Attrib
3 @RT(0) @RT(0) @RT(0)
@END_Attrib
1 0 @F @F @F @F

@END_Dcl

@END_Export

@BEG_Body
@TL(37)
(**************************************** WARNING ********************************************
 *** The KEBA Kemro K2 System including software is not intended for safety control tasks! ***
 ***                       For further information see Comment tab!                        ***
 *********************************************************************************************)

mpbButtonGeneralFwd := EMPTY;
mpbButtonGeneralBwd := EMPTY;

mbDIButtonFwdLinked := IS_LINKED(di_ButtonFwd);
mbDIButtonBwdLinked := IS_LINKED(di_ButtonBwd);

mbDIButtonGeneralFwdLinked := IS_LINKED(di_ButtonGeneral2);
mbDIButtonGeneralBwdLinked := IS_LINKED(di_ButtonGeneral1);

IF (mbDIButtonGeneralFwdLinked AND mbDIButtonGeneralBwdLinked) THEN
    mpiPanelMovementSelector := @sv_iPanelMovementSelector;
END_IF;

// register combinded fwd/bwd button
evPanelButtonRegisterData.Button.nPanelButtonType := nPanelButtonMovement;
evPanelButtonRegisterData.Button.iCompId := sv_DeviceId.CompId;
evPanelButtonRegisterData.Button.iIndexId := sv_DeviceId.IndexId;
evPanelButtonRegisterData.Button.iButtonId := cButtonMoveFwdBwd;
evPanelButtonRegisterData.Button.pbActionVar1 := @sv_bButtonBwd;
evPanelButtonRegisterData.Button.pbActionVar2 := @sv_bButtonFwd;
evPanelButtonRegisterData.Button.Optional.pbLimitSwitch1:= @sv_bEjectorBwd;
evPanelButtonRegisterData.Button.Optional.pbLimitSwitch2:= @sv_bEjectorFwd;
IF sv_bTransducerAvailable THEN
   evPanelButtonRegisterData.Button.Optional.prActVar := @sv_rEjectorPositionRel;
END_IF;
evPanelButtonRegisterData.Button.Optional.prMaxVar := @sv_rEjectorStroke;
evPanelButtonRegisterData.Button.Optional.prMinVar := EMPTY;
evPanelButtonRegisterData.Button.Optional.iBarAttr := 0;

SET_EVENT(evPanelButtonRegister, evPanelButtonRegisterData);

@END_Body

@@@BEG_Comment@@@
@TL(0)

@@@END_Comment@@@

@BEG_Body
@TL(20)
(**************************************** WARNING ********************************************
 *** The KEBA Kemro K2 System including software is not intended for safety control tasks! ***
 ***                       For further information see Comment tab!                        ***
 *********************************************************************************************)

// soft panel button
bButton := sv_bButtonFwd;

// hw panel button
IF mbDIButtonFwdLinked THEN
    bButton := bButton OR di_ButtonFwd;
END_IF;

// external panel button
IF CHECK_REF(mpbButtonGeneralFwd^) THEN
    bButton := bButton OR mpbButtonGeneralFwd^;
END_IF;

abManualButton.aButtonFwd(bButtonFwd := bButton);

@END_Body

@@@BEG_Comment@@@
@TL(0)

@@@END_Comment@@@

@BEG_Body
@TL(21)
(**************************************** WARNING ********************************************
 *** The KEBA Kemro K2 System including software is not intended for safety control tasks! ***
 ***                       For further information see Comment tab!                        ***
 *********************************************************************************************)

// soft panel button
bButton := sv_bButtonBwd;

// hw panel button
IF mbDIButtonBwdLinked THEN
    bButton := bButton OR di_ButtonBwd;
END_IF;

// external panel button
IF CHECK_REF(mpbButtonGeneralBwd^) THEN
    bButton := bButton OR mpbButtonGeneralBwd^;
END_IF;

abManualButton.aButtonBwd(bButtonBwd := bButton);

@END_Body

@@@BEG_Comment@@@
@TL(0)

@@@END_Comment@@@

@BEG_Body
@TL(27)
(**************************************** WARNING ********************************************
 *** The KEBA Kemro K2 System including software is not intended for safety control tasks! ***
 ***                       For further information see Comment tab!                        ***
 *********************************************************************************************)
mpbButtonGeneralFwd := EMPTY;
mpbButtonGeneralBwd := EMPTY;

IF (NOT sv_bDeviceReady) THEN
    // stop active movements
    abManualButton.aButtonFwd(bButtonFwd := FALSE);
    abManualButton.aButtonBwd(bButtonBwd := FALSE);
END_IF;

IF (sv_iPanelMovementSelector > 0) THEN
    Button := sv_PanelButtons[sv_iPanelMovementSelector];
    IF (Button.iCompId = sv_DeviceId.CompId AND
        Button.iIndexId = sv_DeviceId.IndexId) THEN
        IF (Button.iButtonId = cButtonMoveFwdBwd) THEN
            mpbButtonGeneralFwd := @di_ButtonGeneral2;
            mpbButtonGeneralBwd := @di_ButtonGeneral1;
        END_IF;
    END_IF;
END_IF;

@END_Body

@@@BEG_Comment@@@
@TL(0)

@@@END_Comment@@@
@END_Body

@END_Contents

(* ---- ABCheckEjectorMode.pu ---- *)
(*
@h    ! WARNING !
@h    The Kemro K2 system (including software) only meets category B according to EN 954-1,
@h    thus it is not intended for usage in safety-relevant control applications in the field
@h    of personal safety (e.g. emergency stop).
@h    To implement potentially necessary safety-relevant control tasks, always use additional
@h    external safety devices that are intended for the particular purpose, and meet the necessary
@h    functional safety.
@h    For further information see EN 954-1 (EN ISO 13849-1) and/or the K2-x00 user manual, chapter
@h    "CE conformity, directives and standards".

lock full automatic mode when "ejector hold" mode is selected
*)

IMPORT_OVER_LISTFILE
 cCompOperationMode
, tnEjectorMode
, tnOperationMode
, ALARM_EVENT
, FBLockUnlock
, tsAlarm
, ALARM_EVENT_DATA

END_IMPORT

ALGORITHM_BLOCK ABCheckEjectorMode #DUMMY_EDIT_BLOCK

SYSTEM_VAR
 sv_EjectorMode : tnEjectorMode;
 sv_bInitDone : BOOL;
 sv_OperationMode : tnOperationMode;
 sv_bUseProgramSwitches : BOOL;
END_VAR

SYSTEM_OBJECT
 erEjectorHoldInFA : ALARM;
 PU_Task_7 : TASK;
 evAlarmAutoHalf : ALARM_EVENT;
END_OBJECT

POSTUPDATE_ALGORITHM pEjeModeChanged ON PU_Task_7 WITH sv_EjectorMode,sv_bInitDone,sv_bUseProgramSwitches

VAR
 fbLockUnlockOpMode : FBLockUnlock;
 Alarm : tsAlarm;
 bInitDone : BOOL;
 null : ALARM_EVENT_DATA;
END_VAR
#BEGIN_EDIT_BLOCK
(**************************************** WARNING ********************************************
 *** The KEBA Kemro K2 System including software is not intended for safety control tasks! ***
 ***                       For further information see Comment tab!                        ***
 *********************************************************************************************)

IF NOT bInitDone THEN
    fbLockUnlockOpMode.DeviceId.CompId := cCompOperationMode;
    fbLockUnlockOpMode.DeviceId.IndexId := 1;
    Alarm.AlarmId := erEjectorHoldInFA;
    bInitDone := TRUE;
END_IF;

IF (sv_EjectorMode = nHold) AND sv_bUseProgramSwitches THEN
    //full automatic not allowed if hold mode is selected
    fbLockUnlockOpMode.Mode := nLockAbort;
    IF sv_OperationMode = nFullAutomatic THEN
        SET_ALARM(erEjectorHoldInFA);
        SET_EVENT(evAlarmAutoHalf, null);
    END_IF;
ELSE
    //allow change to full automatic
    fbLockUnlockOpMode.Mode := nUnlock;
END_IF;

fbLockUnlockOpMode(MoveDir := cModeFullAutomatic,
                   MoveId := cModeFullAutomatic,
                   Alarm := Alarm);

;#END_EDIT_BLOCK END_ALGORITHM

END_ALGORITHM_BLOCK

#END_OF_IEC_PART

@Puma @IecEditor 6 80 @Pou 25
@@@BEG_Comment@@@
@h    ! WARNING !
@h    The Kemro K2 system (including software) only meets category B according to EN 954-1,
@h    thus it is not intended for usage in safety-relevant control applications in the field
@h    of personal safety (e.g. emergency stop).
@h    To implement potentially necessary safety-relevant control tasks, always use additional
@h    external safety devices that are intended for the particular purpose, and meet the necessary
@h    functional safety.
@h    For further information see EN 954-1 (EN ISO 13849-1) and/or the K2-x00 user manual, chapter
@h    "CE conformity, directives and standards".

lock full automatic mode when "ejector hold" mode is selected
@@@END_Comment@@@

@BEG_Contents

@BEG_Func
@RT(17)FuncTreeContainer
0
@END_Func

@BEG_Const
@RT(18)ConstTreeContainer
1
@Var @RT(18)cCompOperationMode @RT(0) @T @F @DT @RT(4)DINT @RT(0) @T @T @BASIC 0 @F
@F @F
@T
@BEG_Attrib
0 @RT(3)111 @RT(24)Component Operation Mode
@END_Attrib
1 1 @F @F @F @F

@END_Const

@BEG_Export

@BEG_Kind
@ALGORITHM_BLOCK @RT(18)ABCheckEjectorMode @STRUCTURED_TEXT
@RT(0) @RT(0) @RT(0)
@END_Kind

@BEG_Dcl
@RT(16)DclTreeContainer
7
@Var @RT(14)sv_EjectorMode @RT(0) @T @T @RENAMED 0 @T @T @DT @RT(13)tnEjectorMode @RT(0) @T @T @UNKNOWN 0 @F
@F @F
@T
@BEG_Attrib
3 @RT(0) @RT(0) @RT(0)
@END_Attrib
1 8 @F @F @F @F

@Var @RT(17)erEjectorHoldInFA @RT(0) @T @F @DT @RT(5)ALARM @RT(0) @T @T @BASIC 0 @F
@F @F
@T
@BEG_Attrib
3 @RT(0) @RT(0) @RT(0)
@END_Attrib
1 7 @F @F @F @F

@Var @RT(9)PU_Task_7 @RT(0) @T @F @DT @RT(4)TASK @RT(0) @T @T @BASIC 0 @F
@F @F
@T
@BEG_Attrib
3 @RT(0) @RT(0) @RT(0)
@END_Attrib
1 7 @F @F @F @F

@Var @RT(12)sv_bInitDone @RT(0) @T @F @DT @RT(4)BOOL @RT(0) @T @T @BASIC 0 @F
@F @F
@T
@BEG_Attrib
3 @RT(0) @RT(0) @RT(0)
@END_Attrib
1 8 @F @F @F @F

@Var @RT(16)sv_OperationMode @RT(0) @T @T @DERIVED 0 @T @T @DT @RT(15)tnOperationMode @RT(0) @T @T @UNKNOWN 0 @F
@F @F
@T
@BEG_Attrib
3 @RT(0) @RT(0) @RT(0)
@END_Attrib
1 8 @F @F @F @F

@Var @RT(15)evAlarmAutoHalf @RT(0) @T @T @DERIVED 0 @T @T @DT @RT(11)ALARM_EVENT @RT(0) @T @T @UNKNOWN 0 @F
@F @F
@T
@BEG_Attrib
3 @RT(0) @RT(0) @RT(0)
@END_Attrib
1 7 @F @F @F @F

@Var @RT(22)sv_bUseProgramSwitches @RT(0) @T @T @RENAMED 0 @T @T @DT @RT(4)BOOL @RT(0) @T @T @BASIC 0 @F
@F @F
@T
@BEG_Attrib
3 @RT(0) @RT(0) @RT(0)
@END_Attrib
1 8 @F @F @F @F

@END_Dcl

@END_Export

@BEG_Body

1

@BEG_Export

@BEG_Algo
@POSTUPDATE_ALGORITHM @RT(15)pEjeModeChanged @STRUCTURED_TEXT
@RT(0) @RT(50)sv_EjectorMode,sv_bInitDone,sv_bUseProgramSwitches @RT(9)PU_Task_7 @F @F
@END_Algo

@BEG_Dcl
@RT(16)DclTreeContainer
4
@Var @RT(18)fbLockUnlockOpMode @RT(0) @T @T @DERIVED 0 @T @T @DT @RT(12)FBLockUnlock @RT(0) @T @T @UNKNOWN 0 @F
@F @F
@T
@BEG_Attrib
3 @RT(0) @RT(0) @RT(0)
@END_Attrib
1 0 @F @F @F @F

@Var @RT(5)Alarm @RT(0) @T @T @DERIVED 0 @T @T @DT @RT(7)tsAlarm @RT(0) @T @T @UNKNOWN 0 @F
@F @F
@T
@BEG_Attrib
3 @RT(0) @RT(0) @RT(0)
@END_Attrib
1 0 @F @F @F @F

@Var @RT(9)bInitDone @RT(0) @T @F @DT @RT(4)BOOL @RT(0) @T @T @BASIC 0 @F
@F @F
@T
@BEG_Attrib
3 @RT(0) @RT(0) @RT(0)
@END_Attrib
1 0 @F @F @F @F

@Var @RT(4)null @RT(0) @T @T @DERIVED 0 @T @T @DT @RT(16)ALARM_EVENT_DATA @RT(0) @T @T @UNKNOWN 0 @F
@F @F
@T
@BEG_Attrib
3 @RT(0) @RT(0) @RT(0)
@END_Attrib
1 0 @F @F @F @F

@END_Dcl

@END_Export

@BEG_Body
@TL(29)
(**************************************** WARNING ********************************************
 *** The KEBA Kemro K2 System including software is not intended for safety control tasks! ***
 ***                       For further information see Comment tab!                        ***
 *********************************************************************************************)

IF NOT bInitDone THEN
    fbLockUnlockOpMode.DeviceId.CompId := cCompOperationMode;
    fbLockUnlockOpMode.DeviceId.IndexId := 1;
    Alarm.AlarmId := erEjectorHoldInFA;
    bInitDone := TRUE;
END_IF;

IF (sv_EjectorMode = nHold) AND sv_bUseProgramSwitches THEN
    //full automatic not allowed if hold mode is selected
    fbLockUnlockOpMode.Mode := nLockAbort;
    IF sv_OperationMode = nFullAutomatic THEN
        SET_ALARM(erEjectorHoldInFA);
        SET_EVENT(evAlarmAutoHalf, null);
    END_IF;
ELSE
    //allow change to full automatic
    fbLockUnlockOpMode.Mode := nUnlock;
END_IF;

fbLockUnlockOpMode(MoveDir := cModeFullAutomatic,
                   MoveId := cModeFullAutomatic,
                   Alarm := Alarm);

@END_Body

@@@BEG_Comment@@@
@TL(0)

@@@END_Comment@@@
@END_Body

@END_Contents

(* ---- ABDefaultConditions.pu ---- *)
(*
@h    ! WARNING !
@h    The Kemro K2 system (including software) only meets category B according to EN 954-1,
@h    thus it is not intended for usage in safety-relevant control applications in the field
@h    of personal safety (e.g. emergency stop).
@h    To implement potentially necessary safety-relevant control tasks, always use additional
@h    external safety devices that are intended for the particular purpose, and meet the necessary
@h    functional safety.
@h    For further information see EN 954-1 (EN ISO 13849-1) and/or the K2-x00 user manual, chapter
@h    "CE conformity, directives and standards".

This AB monitors following default conditions:
If the ejector is not bwd, all mold close movements are locked.
If the ejector is not bwd, all core movements are locked.

This default conditions are not monitored in the following cases:
+ The machine sequence is created by machine sequencer and not by ODC - files
+ monitoring is deactivated (sv_bIgnoreDefaultConditions = TRUE)
+ If "override core safety" is activated, the ejector position has no influence on core movements.

*)

IMPORT_OVER_LISTFILE
 cCompCore
, FBLockUnlock
, KSYS_Status

END_IMPORT

ALGORITHM_BLOCK ABDefaultConditions #DUMMY_EDIT_BLOCK

SYSTEM_VAR
 sv_bEjectorBwd : BOOL;
 sv_bInitDone : BOOL;
 sv_bInitStart : BOOL;
 sv_bIgnoreDefaultConditions : BOOL;
 sv_bOverrideCoreSafety : BOOL;
 sv_bUseProgramSwitches : BOOL;
END_VAR

SYSTEM_OBJECT
 PU_Task_7 : TASK;
 erEjectorNotBackward : ALARM;
 PU_Task_3 : TASK;
END_OBJECT

VAR
 mpiNewSequence : REFTO DINT;
END_VAR

ALGORITHM aLockUnlock

VAR
 fbLockUnlock : FBLockUnlock;
END_VAR
#BEGIN_EDIT_BLOCK
(**************************************** WARNING ********************************************
 *** The KEBA Kemro K2 System including software is not intended for safety control tasks! ***
 ***                       For further information see Comment tab!                        ***
 *********************************************************************************************)

IF NOT sv_bInitDone THEN
   RETURN;  //no lock / unlock before sv_bInitDone
END_IF;

IF sv_bIgnoreDefaultConditions OR NOT sv_bUseProgramSwitches THEN
   //sequence programmmed by machine sequencer or
   //default conditions deactivated
   fbLockUnlock.Mode := nUnlock;
ELSE
   //sequence programmed by files and default conditions activated
   //-> check default conditions
   IF sv_bEjectorBwd THEN
      fbLockUnlock.Mode := nUnlock;
   ELSE
      fbLockUnlock.Mode := nLockAbort;
   END_IF;
END_IF;

//lock /unlock mold close
fbLockUnlock.DeviceId.CompId := cCompMold;
fbLockUnlock.DeviceId.IndexId := 1;
fbLockUnlock.MoveDir := cMoveFwd;
fbLockUnlock.MoveId := cMoveAll;
fbLockUnlock.Alarm.AlarmId := erEjectorNotBackward;
fbLockUnlock();

//lock / unlock all core movements if ejector is not bwd
//also consider "override core safety"
IF sv_bOverrideCoreSafety THEN
   fbLockUnlock.Mode := nUnlock;
END_IF;
fbLockUnlock.DeviceId.CompId := cCompCore;
fbLockUnlock.DeviceId.IndexId := cAllDevIndex;
fbLockUnlock.MoveDir := cMoveAll;
fbLockUnlock.MoveId := cMoveAll;
fbLockUnlock.Alarm.AlarmId := erEjectorNotBackward;
fbLockUnlock();

;#END_EDIT_BLOCK END_ALGORITHM

POSTUPDATE_ALGORITHM pInitStart ON PU_Task_7 WITH sv_bInitStart

VAR
 state : KSYS_Status;
END_VAR
#BEGIN_EDIT_BLOCK
(**************************************** WARNING ********************************************
 *** The KEBA Kemro K2 System including software is not intended for safety control tasks! ***
 ***                       For further information see Comment tab!                        ***
 *********************************************************************************************)

//get reference
mpiNewSequence := GET_SYNC_REFTO('ODC1.sv_iODCSequenceUpdated', T#0s, state);

;#END_EDIT_BLOCK END_ALGORITHM

POSTUPDATE_ALGORITHM pCheckDefaultConditions ON PU_Task_3 WITH sv_bEjectorBwd,mpiNewSequence^,sv_bIgnoreDefaultConditions,sv_bOverrideCoreSafety

#BEGIN_EDIT_BLOCK
(**************************************** WARNING ********************************************
 *** The KEBA Kemro K2 System including software is not intended for safety control tasks! ***
 ***                       For further information see Comment tab!                        ***
 *********************************************************************************************)

aLockUnlock();

;#END_EDIT_BLOCK END_ALGORITHM

END_ALGORITHM_BLOCK

#END_OF_IEC_PART

@Puma @IecEditor 6 126 @Pou 25
@@@BEG_Comment@@@
@h    ! WARNING !
@h    The Kemro K2 system (including software) only meets category B according to EN 954-1,
@h    thus it is not intended for usage in safety-relevant control applications in the field
@h    of personal safety (e.g. emergency stop).
@h    To implement potentially necessary safety-relevant control tasks, always use additional
@h    external safety devices that are intended for the particular purpose, and meet the necessary
@h    functional safety.
@h    For further information see EN 954-1 (EN ISO 13849-1) and/or the K2-x00 user manual, chapter
@h    "CE conformity, directives and standards".

This AB monitors following default conditions:
If the ejector is not bwd, all mold close movements are locked.
If the ejector is not bwd, all core movements are locked.

This default conditions are not monitored in the following cases:
+ The machine sequence is created by machine sequencer and not by ODC - files
+ monitoring is deactivated (sv_bIgnoreDefaultConditions = TRUE)
+ If "override core safety" is activated, the ejector position has no influence on core movements.

@@@END_Comment@@@

@BEG_Contents

@BEG_Func
@RT(17)FuncTreeContainer
0
@END_Func

@BEG_Const
@RT(18)ConstTreeContainer
1
@Var @RT(9)cCompCore @RT(0) @T @F @DT @RT(4)DINT @RT(0) @T @T @BASIC 0 @F
@F @F
@T
@BEG_Attrib
0 @RT(3)109 @RT(14)Component Core
@END_Attrib
1 1 @F @F @F @F

@END_Const

@BEG_Export

@BEG_Kind
@ALGORITHM_BLOCK @RT(19)ABDefaultConditions @STRUCTURED_TEXT
@RT(0) @RT(0) @RT(0)
@END_Kind

@BEG_Dcl
@RT(16)DclTreeContainer
10
@Var @RT(9)PU_Task_7 @RT(0) @T @T @RENAMED 0 @T @T @DT @RT(4)TASK @RT(0) @T @T @BASIC 0 @F
@F @F
@T
@BEG_Attrib
3 @RT(0) @RT(0) @RT(0)
@END_Attrib
1 7 @F @F @F @F

@Var @RT(14)sv_bEjectorBwd @RT(0) @T @T @RENAMED 0 @T @T @DT @RT(4)BOOL @RT(0) @T @T @BASIC 0 @F
@F @F
@T
@BEG_Attrib
3 @RT(0) @RT(0) @RT(0)
@END_Attrib
1 8 @F @F @F @F

@Var @RT(20)erEjectorNotBackward @RT(0) @T @F @DT @RT(5)ALARM @RT(0) @T @T @BASIC 0 @F
@F @F
@T
@BEG_Attrib
3 @RT(0) @RT(0) @RT(0)
@END_Attrib
1 7 @F @F @F @F

@Var @RT(12)sv_bInitDone @RT(0) @T @T @RENAMED 0 @T @T @DT @RT(4)BOOL @RT(0) @T @T @BASIC 0 @F
@F @F
@T
@BEG_Attrib
3 @RT(0) @RT(0) @RT(0)
@END_Attrib
1 8 @F @F @F @F

@Var @RT(13)sv_bInitStart @RT(0) @T @T @RENAMED 0 @T @T @DT @RT(4)BOOL @RT(0) @T @T @BASIC 0 @F
@F @F
@T
@BEG_Attrib
3 @RT(0) @RT(0) @RT(0)
@END_Attrib
1 8 @F @F @F @F

@Var @RT(14)mpiNewSequence @RT(0) @T @T @REFTO 0 @T @DT @RT(4)DINT @RT(0) @T @T @BASIC 0 @F
@F @F
@T
@BEG_Attrib
3 @RT(0) @RT(0) @RT(0)
@END_Attrib
1 0 @F @F @F @F

@Var @RT(27)sv_bIgnoreDefaultConditions @RT(0) @T @T @RENAMED 0 @T @T @DT @RT(4)BOOL @RT(0) @T @T @BASIC 0 @F
@F @F
@T
@BEG_Attrib
3 @RT(0) @RT(0) @RT(0)
@END_Attrib
1 8 @F @F @F @F

@Var @RT(22)sv_bOverrideCoreSafety @RT(0) @T @T @RENAMED 0 @T @T @DT @RT(4)BOOL @RT(0) @T @T @BASIC 0 @F
@F @F
@T
@BEG_Attrib
3 @RT(0) @RT(0) @RT(0)
@END_Attrib
1 8 @F @F @F @F

@Var @RT(22)sv_bUseProgramSwitches @RT(0) @T @F @DT @RT(4)BOOL @RT(0) @T @T @BASIC 0 @F
@F @F
@T
@BEG_Attrib
3 @RT(0) @RT(0) @RT(0)
@END_Attrib
1 8 @F @F @F @F

@Var @RT(9)PU_Task_3 @RT(0) @T @T @RENAMED 0 @T @T @DT @RT(4)TASK @RT(0) @T @T @BASIC 0 @F
@F @F
@T
@BEG_Attrib
3 @RT(0) @RT(0) @RT(0)
@END_Attrib
1 7 @F @F @F @F

@END_Dcl

@END_Export

@BEG_Body

3

@BEG_Export

@BEG_Algo
@ALGORITHM @RT(11)aLockUnlock @STRUCTURED_TEXT
@RT(0) @RT(0) @RT(0) @F @F
@END_Algo

@BEG_Dcl
@RT(16)DclTreeContainer
1
@Var @RT(12)fbLockUnlock @RT(0) @T @T @DERIVED 0 @T @T @DT @RT(12)FBLockUnlock @RT(0) @T @T @UNKNOWN 0 @F
@F @F
@T
@BEG_Attrib
3 @RT(0) @RT(0) @RT(0)
@END_Attrib
1 0 @F @F @F @F

@END_Dcl

@END_Export

@BEG_Export

@BEG_Algo
@POSTUPDATE_ALGORITHM @RT(10)pInitStart @STRUCTURED_TEXT
@RT(0) @RT(13)sv_bInitStart @RT(9)PU_Task_7 @F @F
@END_Algo

@BEG_Dcl
@RT(16)DclTreeContainer
1
@Var @RT(5)state @RT(0) @T @T @DERIVED 0 @T @T @DT @RT(11)KSYS_Status @RT(0) @T @T @UNKNOWN 0 @F
@F @F
@T
@BEG_Attrib
3 @RT(0) @RT(0) @RT(0)
@END_Attrib
1 0 @F @F @F @F

@END_Dcl

@END_Export

@BEG_Export

@BEG_Algo
@POSTUPDATE_ALGORITHM @RT(23)pCheckDefaultConditions @STRUCTURED_TEXT
@RT(0) @RT(81)sv_bEjectorBwd,mpiNewSequence^,sv_bIgnoreDefaultConditions,sv_bOverrideCoreSafety @RT(9)PU_Task_3 @F @F
@END_Algo

@BEG_Dcl
@RT(16)DclTreeContainer
0
@END_Dcl

@END_Export

@BEG_Body
@TL(45)
(**************************************** WARNING ********************************************
 *** The KEBA Kemro K2 System including software is not intended for safety control tasks! ***
 ***                       For further information see Comment tab!                        ***
 *********************************************************************************************)

IF NOT sv_bInitDone THEN
   RETURN;  //no lock / unlock before sv_bInitDone
END_IF;

IF sv_bIgnoreDefaultConditions OR NOT sv_bUseProgramSwitches THEN
   //sequence programmmed by machine sequencer or
   //default conditions deactivated
   fbLockUnlock.Mode := nUnlock;
ELSE
   //sequence programmed by files and default conditions activated
   //-> check default conditions
   IF sv_bEjectorBwd THEN
      fbLockUnlock.Mode := nUnlock;
   ELSE
      fbLockUnlock.Mode := nLockAbort;
   END_IF;
END_IF;

//lock /unlock mold close
fbLockUnlock.DeviceId.CompId := cCompMold;
fbLockUnlock.DeviceId.IndexId := 1;
fbLockUnlock.MoveDir := cMoveFwd;
fbLockUnlock.MoveId := cMoveAll;
fbLockUnlock.Alarm.AlarmId := erEjectorNotBackward;
fbLockUnlock();

//lock / unlock all core movements if ejector is not bwd
//also consider "override core safety"
IF sv_bOverrideCoreSafety THEN
   fbLockUnlock.Mode := nUnlock;
END_IF;
fbLockUnlock.DeviceId.CompId := cCompCore;
fbLockUnlock.DeviceId.IndexId := cAllDevIndex;
fbLockUnlock.MoveDir := cMoveAll;
fbLockUnlock.MoveId := cMoveAll;
fbLockUnlock.Alarm.AlarmId := erEjectorNotBackward;
fbLockUnlock();

@END_Body

@@@BEG_Comment@@@
@TL(0)

@@@END_Comment@@@

@BEG_Body
@TL(8)
(**************************************** WARNING ********************************************
 *** The KEBA Kemro K2 System including software is not intended for safety control tasks! ***
 ***                       For further information see Comment tab!                        ***
 *********************************************************************************************)

//get reference
mpiNewSequence := GET_SYNC_REFTO('ODC1.sv_iODCSequenceUpdated', T#0s, state);

@END_Body

@@@BEG_Comment@@@
@TL(0)

@@@END_Comment@@@

@BEG_Body
@TL(7)
(**************************************** WARNING ********************************************
 *** The KEBA Kemro K2 System including software is not intended for safety control tasks! ***
 ***                       For further information see Comment tab!                        ***
 *********************************************************************************************)

aLockUnlock();

@END_Body

@@@BEG_Comment@@@
@TL(0)

@@@END_Comment@@@
@END_Body

@END_Contents
